Staubli VAL3: onF6Event.pgx

program onF6Event(bool& x_bSave[])
  local string l_sName
  local num l_nResult
  local string l_sSwap
  local string l_sMessage
  local bool l_bYes
  local string l_sButton[2]
begin
  // look if the bButton is enable
  if bButton[5]
    //
    // delete the selected ITEM
    //
    call axis:get(l_sName,nIndex)
    if l_sName=="workPos"
      call use:timerDialog("该点为系统所有，无法删除",1)
      return
    endIf

    if nIndex>=0
      call axis:get(l_sName,nIndex)
      if l_sName!=""
        l_sSwap=l_sName="AXIS8>"+l_sName

        if l_nResult==0

          if l_nResult==0
            //delete it
            call language:message(l_sMessage,80)
            call language:getYesNo(l_sButton)
            call use:yes_no(l_sMessage,l_sButton,l_bYes)
            if l_bYes
              call axis:del(nIndex)
              logMsg("[KERNEL] INTERFACE:Delete the AXIS8: "+sEvent+" at position: "+toString("",nIndex))
              // for the refresh
              if nIndex>0
                nIndex=nIndex-1
                if nIndex<nView
                  nView=nIndex
                endIf
              endIf
              nSelected=nIndex
              call buildList()
              call refreshStatic()
              // save it
              x_bSave=true
            endIf
          endIf
        endIf
        if l_nResult!=0
          // TODO
          call showExist(l_sName,l_sSwap)
        endIf
      endIf
    endIf
  endIf

end
